// TIA Portal V20 export
DATA_BLOCK "BK01"   // DB298
// stored: Access Published, MemoryReserve 100
   VAR
      "X10-1 JR OUT P&P1 Y-AXIS ROBOT LIMIT SENSOR(-)" : Bool;
      "X11-1 JR OUT P&P1 Y-AXIS ROBOT LIMIT SENSOR(+)" : Bool;
      "X12-1 JR OUT P&P2 Y-AXIS ROBOT LIMIT SENSOR(-)" : Bool;
      "X13-1 JR OUT P&P2 Y-AXIS ROBOT LIMIT SENSOR(+)" : Bool;
      "X14-1 STACK 1 NG BOX DETECT SENSOR" : Bool;
      "X15-1 SPARE" : Bool;
      "X16-1 SPARE" : Bool;
      "X17-1 SPARE" : Bool;
      "X10-2 JR OUT P&P1 Y-AXIS ROBOT HOME SENSOR" : Bool;
      "X11-2 SPARE" : Bool;
      "X12-2 JR OUT P&P2 Y-AXIS ROBOT HOME SENSOR" : Bool;
      "X13-2 SPARE" : Bool;
      "X14-2 STACK 2 NG BOX DETECT SENSOR" : Bool;
      "X15-2 SPARE" : Bool;
      "X16-2 SPARE" : Bool;
      "X17-2 SPARE" : Bool;
   END_VAR
BEGIN
END_DATA_BLOCK
